FUNCTION_BLOCK FB_SerialComRS232
VAR_IN_OUT

	stEL6001In : EL6inData22B;
	stEL6001Out : EL6outData22B;
END_VAR
VAR_OUTPUT
	aAcceleration : ARRAY [0..2] OF REAL;
	eReceiveErrorID	: ComError_t;
	nReceiveCounter	: UDINT;
END_VAR
VAR

	//Receive Buffer
	fbEL6001Ctrl		: SerialLineControl;
	TxBuffer	: ComBuffer;
	RxBuffer	: ComBuffer;
	//Receive Data
	fbReceive		: ReceiveData;
	nPrefix : ARRAY[0..1] OF BYTE;
	aReceiveData : ARRAY [0..15] OF BYTE;
	nPacketID : BYTE := 37;
	nPacketLength : BYTE := 12;	
	
	nCRC : WORD;
	nCheckCRC : WORD;
	nPointerCRC : POINTER TO WORD;
	aCRC : ARRAY [0..1] OF BYTE;	
	aDataArray : ARRAY[0..11] OF BYTE;
	i : USINT;
	aAccX : ARRAY [0..3] OF BYTE;
	aAccY : ARRAY [0..3] OF BYTE;
	aAccZ : ARRAY [0..3] OF BYTE;
	fPointerToX : POINTER TO REAL;
    fAccX : REAL;
	fPointerToY : POINTER TO REAL;
    fAccY : REAL;
	fPointerToZ : POINTER TO REAL;
    fAccZ : REAL;
END_VAR

fbEL6001Ctrl(
	Mode:= SERIALLINEMODE_EL6_22B, 
	pComIn:= ADR(stEL6001In), 
	pComOut:= ADR(stEL6001Out), 
	SizeComIn:= SIZEOF(stEL6001In), 
	Error=> , 
	ErrorID=> , 
	TxBuffer:= TxBuffer, 
	RxBuffer:= RxBuffer);

nPrefix[0] := nPacketID;
nPrefix[1] := nPacketLength;

fbReceive(
	RXbuffer:= RxBuffer,
	pPrefix := ADR(nPrefix),
	LenPrefix := 2,
	pReceiveData := ADR(aReceiveData),
	SizeReceiveData  := 16,								
	Error => eReceiveErrorID,
	DataReceived=>);
		
IF fbReceive.DataReceived THEN							
	nReceiveCounter := nReceiveCounter + 1;
END_IF

doCRC16Check();
doCalculateAccValues();

METHOD PRIVATE doCalculateAccValues
VAR_INPUT
END_VAR
IF nCheckCRC = nCRC THEN
	aAccX[0] := aReceiveData[4];
	aAccX[1] := aReceiveData[5];
	aAccX[2] := aReceiveData[6];
	aAccX[3] := aReceiveData[7];
	fPointerToX := ADR(aAccX);
	fAccX := fPointerToX^;
	
	aAccY[0] := aReceiveData[8];
	aAccY[1] := aReceiveData[9];
	aAccY[2] := aReceiveData[10];
	aAccY[3] := aReceiveData[11];
	fPointerToY := ADR(aAccY);
	fAccY := fPointerToY^;
	
	aAccZ[0] := aReceiveData[12];
	aAccZ[1] := aReceiveData[13];
	aAccZ[2] := aReceiveData[14];
	aAccZ[3] := aReceiveData[15];
	fPointerToZ := ADR(aAccZ);
	fAccZ := fPointerToZ^;
END_IF

aAcceleration[0] := fAccX;
aAcceleration[1] := fAccY;
aAcceleration[2] := fAccZ;
END_METHOD

METHOD PRIVATE doCRC16Check : BOOL
VAR_INPUT
END_VAR
FOR i:=0 TO 11 DO
	aDataArray[i] := aReceiveData[i+4];
END_FOR


nCRC := F_DATA_TO_CRC16_CCITT(
	pData := ADR(aDataArray),
	cbData := BYTE_TO_UDINT(nPacketLength),
	crc := 16#FFFF);

aCRC[0] := aReceiveData[2];
aCRC[1] := aReceiveData[3];
nPointerCRC := ADR(aCRC);
nCheckCRC := nPointerCRC^;
END_METHOD

END_FUNCTION_BLOCK

(* stored: Version 1.1.0.1, ProductVersion 3.1.4024.12
   POU FB_SerialComRS232: Id {9d3d8819-cac2-416e-a680-ea14d4dc7b50}, SpecialFunc None
   Method doCalculateAccValues: Id {752dfdc0-a0a9-4925-a6a6-e26264e0e3c3}
   Method doCRC16Check: Id {4d6586cc-d4c5-4d49-a10a-4faa26ac239a} *)
